(* IEC 61131-3 sources: IEC61131-3-CDSV3/PCRE2/src/Native, 9 files *)

(* ---- FuCompilePCRE_cext.pou ---- *)
(*#-#-#-#-#-#-#-#-#-#---Declaration---#-#-#-#-#-#-#-#-#-#-#-#-#*)

{attribute 'qualified_only'}
FUNCTION INTERNAL FuCompilePCRE_cext : __XWORD
VAR_INPUT
    psPattern: POINTER TO STRING(1);
    udiLength: UDINT;
    udiOptions: UDINT;
END_VAR
(*#-#-#-#-#-#-#-#-#-#---Implementation---#-#-#-#-#-#-#-#-#-#-#-#-#*)

; // Nothing to do in simulation mode

(* ---- FuFreeMatchPCRE_cext.pou ---- *)
(*#-#-#-#-#-#-#-#-#-#---Declaration---#-#-#-#-#-#-#-#-#-#-#-#-#*)

{attribute 'qualified_only'}
FUNCTION INTERNAL FuFreeMatchPCRE_cext
VAR_INPUT
    mb: __XWORD;
END_VAR
(*#-#-#-#-#-#-#-#-#-#---Implementation---#-#-#-#-#-#-#-#-#-#-#-#-#*)

; // Nothing to do in simulation mode

(* ---- FuFreePCRE_cext.pou ---- *)
(*#-#-#-#-#-#-#-#-#-#---Declaration---#-#-#-#-#-#-#-#-#-#-#-#-#*)

{attribute 'qualified_only'}
FUNCTION INTERNAL FuFreePCRE_cext
VAR_INPUT
    re: __XWORD;
END_VAR
(*#-#-#-#-#-#-#-#-#-#---Implementation---#-#-#-#-#-#-#-#-#-#-#-#-#*)

; // Nothing to do in simulation mode

(* ---- FuGetMatchPCRE_cext.pou ---- *)
(*#-#-#-#-#-#-#-#-#-#---Declaration---#-#-#-#-#-#-#-#-#-#-#-#-#*)

{attribute 'qualified_only'}
FUNCTION INTERNAL FuGetMatchPCRE_cext : BOOL
VAR_INPUT
    mb: __XWORD;
    psSubject: POINTER TO STRING(1);
    udiSubjectLength: UDINT;
    uiMatchIndex: UINT;
    psMatch: POINTER TO STRING(1);
    udiSize: UDINT;
END_VAR
VAR_OUTPUT
    udiLength: UDINT;
END_VAR
(*#-#-#-#-#-#-#-#-#-#---Implementation---#-#-#-#-#-#-#-#-#-#-#-#-#*)

; // Nothing to do in simulation mode

(* ---- FuGetMatchSubstringLengthPCRE_cext.pou ---- *)
(*#-#-#-#-#-#-#-#-#-#---Declaration---#-#-#-#-#-#-#-#-#-#-#-#-#*)

{attribute 'qualified_only'}
FUNCTION INTERNAL FuGetMatchSubstringLengthPCRE_cext : BOOL
VAR_INPUT
    mb: __XWORD;
    uiMatchIndex: UINT;
END_VAR
VAR_OUTPUT
    udiLength: UDINT;
END_VAR
(*#-#-#-#-#-#-#-#-#-#---Implementation---#-#-#-#-#-#-#-#-#-#-#-#-#*)

; // Nothing to do in simulation mode

(* ---- FuGetNamedMatchPCRE_cext.pou ---- *)
(*#-#-#-#-#-#-#-#-#-#---Declaration---#-#-#-#-#-#-#-#-#-#-#-#-#*)

{attribute 'qualified_only'}
FUNCTION INTERNAL FuGetNamedMatchPCRE_cext : BOOL
VAR_INPUT
    mb: __XWORD;
    psSubject: POINTER TO STRING(1);
    udiSubjectLength: UDINT;
    sMatchName: STRING(255);
    udiMatchIndexLength: UDINT;
    psMatch: POINTER TO STRING(1);
    udiSize: UDINT;
END_VAR
VAR_OUTPUT
    udiLength: UDINT;
END_VAR
(*#-#-#-#-#-#-#-#-#-#---Implementation---#-#-#-#-#-#-#-#-#-#-#-#-#*)

; // Nothing to do in simulation mode

(* ---- FuGetNamedMatchSubstringLengthPCRE_cext.pou ---- *)
(*#-#-#-#-#-#-#-#-#-#---Declaration---#-#-#-#-#-#-#-#-#-#-#-#-#*)

{attribute 'qualified_only'}
FUNCTION INTERNAL FuGetNamedMatchSubstringLengthPCRE_cext : BOOL
VAR_INPUT
    mb: __XWORD;
    sMatchName: STRING(255);
    udiMatchIndexLength: UDINT;
END_VAR
VAR_OUTPUT
    udiLength: UDINT;
END_VAR
(*#-#-#-#-#-#-#-#-#-#---Implementation---#-#-#-#-#-#-#-#-#-#-#-#-#*)

; // Nothing to do in simulation mode

(* ---- FuMatchPCRE_cext.pou ---- *)
(*#-#-#-#-#-#-#-#-#-#---Declaration---#-#-#-#-#-#-#-#-#-#-#-#-#*)

{attribute 'qualified_only'}
FUNCTION INTERNAL FuMatchPCRE_cext : INT
VAR_INPUT
    re: __XWORD;
    psSubject: POINTER TO STRING(1);
    udiLength: UDINT;
    udiOffset: UDINT;
    udiOptions: UDINT;
END_VAR
VAR_OUTPUT
    mb: __XWORD;
END_VAR
(*#-#-#-#-#-#-#-#-#-#---Implementation---#-#-#-#-#-#-#-#-#-#-#-#-#*)

; // Nothing to do in simulation mode

(* ---- FuSimpleMatchPCRE_cext.pou ---- *)
(*#-#-#-#-#-#-#-#-#-#---Declaration---#-#-#-#-#-#-#-#-#-#-#-#-#*)

{attribute 'qualified_only'}
FUNCTION INTERNAL FuSimpleMatchPCRE_cext : BOOL
VAR_INPUT
    re: __XWORD;
    psSubject: POINTER TO STRING(1);
    udiLength: UDINT;
    udiOffset: UDINT;
    udiOptions: UDINT;
END_VAR
(*#-#-#-#-#-#-#-#-#-#---Implementation---#-#-#-#-#-#-#-#-#-#-#-#-#*)

; // Nothing to do in simulation mode
